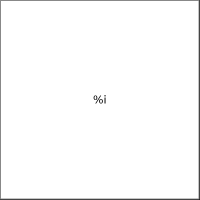
VISUALIZATION Testkachel  // 200x200
VAR_IN_OUT
	FB_DI_16:DI_16;
END_VAR
var_input
	s_Titel:STRING;
END_VAR
    Rectangle (0,0 200x200), "%i", text variable: s_Titel
END_VISUALIZATION

(* stored: Version 1.1.0.1, ProductVersion 3.1.4022.6
   Visu Testkachel: Id {5939df85-be41-4825-80c3-65f9d55afca2} *)
